// SIMATIC S7-200 project (STEP 7-Micro/WIN), CPU 226 REL 01.23

ORGANIZATION_BLOCK 主:OB1
TITLE=PLC通过串行通信与称重传感器交互，获取重量数据，并根据预设标准（重量不得超过100单位）判断产品是否合格。系统确保每个包装袋的重量在规定范围内，避免超重或不足。
// 
// 系统当首次扫描标志为1时，设置通信端口设置为16#09（自由口模式），配置通信起始符为16#54（'T’）、通信结束符为16#0A（换行符）、最大字符数为100，并将设备地址设置为16#03540D0A——这些参数必须正确初始化，否则通信无法正常进行。
// 运行中，当常开标志为1时，接收中断触发，PLC接收数据到缓冲区并设置10毫秒定时中断，随后将数据存入重量数据进行处理，以避免数据丢失。
// 在定时中断中，PLC断开自身中断后，检查重量数据是否大于标准值，并根据结果发送预配置的数据并控制报警输出。若重量数据超标，表明包装袋超重，系统发送数据至上位机并触发报警；否则保持报警关闭，确保报警仅在超重时触发。
// 
BEGIN
Network 1 // 网络标题
// 网络注解
LD     SM0.1
MOVB   16#9, SMB30
MOVB   16#E0, SMB87
MOVB   16#54, SMB88          //起始符
MOVB   16#A, SMB89           //结束字符
MOVB   100, SMB94            //设置最大字符数100
MOVD   16#3540D0A, VD0       //设备地址
ATCH   INT_1:INT1, 23        //接收中断
ATCH   INT_0:INT0, 9         //发送中断
ENI
XMT    VB0, 0                //发送缓冲区VB100  
?000
END_ORGANIZATION_BLOCK

INTERRUPT_BLOCK INT_0:INT0
TITLE=中断例行程序注解
BEGIN
Network 1 // 网络标题
// 网络注解
LD     SM0.0
RCV    VB100, 0
END_INTERRUPT_BLOCK

INTERRUPT_BLOCK INT_1:INT1
TITLE=中断例行程序注解
BEGIN
Network 1 // 网络标题
// 网络注解
LD     SM0.0
MOVB   10, SMB34             // 设置10MS定时, 然后发送
ATCH   INT_2:INT2, 10
CRETI
END_INTERRUPT_BLOCK

INTERRUPT_BLOCK INT_2:INT2
TITLE=中断例行程序注解
BEGIN
Network 1 // 网络标题
// 网络注解
LD     SM0.0                 //10MS 定时中断
DTCH   10                    //断开中断
Network 2
LDD>   VD101, 100
XMT    VB0, 0                // 下一轮地址发送
NOT
=      Q0.0                  //不合格，报警
END_INTERRUPT_BLOCK
